FUNCTION_BLOCK fbChamber
VAR_INPUT
END_VAR
VAR_OUTPUT
END_VAR
VAR_IN_OUT
	stControl				: stControl;
	stInOuts 				: stInOuts;
	stParams				: stParamsChamber;
	stChamberTestParams		: stTestParams;
	stTime					: stAircomTimeStruct;	//Struktura czasu
END_VAR
VAR
	//Bloki skalujące
	fbPressureScaller 		:fbAnalogMeasurement;	//Blok skalujący ciśnienie
	fbVoltageScaller	 	:fbAnalogMeasurement;	//Blok skalujący napięcie
	fbCurrentScaller 		:fbAnalogMeasurement;	//Blok skalujący prąd
	iWorkStep : INT;
	//Detekcja prądu
	fbCurrentCheckDelayer	: TON;					//Zwłoka dla wykrywania prądu minimalnego
	//Test EOL
	fbTestTimerEOL			: TON;					//Licznik czasu trwania testu EOL
	bEolTestResult			: BOOL;					//Wynik z testu EOL
	//Test Performance
	fbTestTimerPerformance	: TON;					//Licznik czasu trwania testu Wydajnoiściowego
	bPerfornamceTestResult	: BOOL;					//Wynik z testu Wydajnościowego
	//Test Hour
	fbTestTimerHour	: TON;							//Licznik czasu trwania testu Wydajnoiściowego
	bHourTestResult	: BOOL;							//Wynik z testu Wydajnościowego
	bPressureObtainedHour :BOOL;					//Pierwsza faza zakończona osiągnięto ciśnienie testowe
	//Test Whole
	iWorkStepWhole	: INT;							//Kroki programowe dla testu całościowego
	fbTestTimerWholeI	: TON;							//Licznik czasu I test całkowity
	fbTestTimerWholeII	: TON;							//Licznik czasu II test całkowity
	//Test Under Presure
	bUnderPresureTestResult : BOOL;					//Wynik testu pod ciśnieniem
	rStartUnderPresureLastPresureRecord : REAL;		//Save value of presure before test
	fbUnderPresureTestTimer	: TON;							//Licznik czasu dla tesu pod ciśnieniem
	//Test Cyclic 30
	iCyclicLoopVariable 		: INT;				//Wariable for calculate of cyclic loops
	fbTestTimerCyclic30			: TON;				//Licznik czasu trwania testu cyklicznego 30
	bCyclic30TestResult			: BOOL;				//Wynik testu cyklicznego x30
	fbTestTimerCyclic30On		: TON;				//Timer dla obsługi testu
	bFirstCycle30				: BOOL;				//First cycle indefiner
	//Test Cyclic 70
	fbTestTimerCyclic70			: TON;				//Licznik czasu trwania testu cyklicznego 30
	bCyclic70TestResult			: BOOL;				//Wynik testu cyklicznego x30
	fbTestTimerCyclic70On		: TON;				//Timer dla obsługi testu
	bFirstCycle70				: BOOL;				//First cycle indefiner
	//Zmienne do obsługi zapisu plików
	sData						: STRING;			//Data dopisana do lokalizacji
	sDate						: STRING;			//Data rozpoczęcia testu
	sTime						: STRING;			//Godzina rozpoczęcia testu
	sTestName					: STRING;			//Nazwa Test
	sFirstLine					: STRING;			//Dane do zapisu w pierwszej linijce
	sDataString					: STRING(5000);			//dane z pomiarami
	sDataStringTmp				: STRING(5000);			//dane z pomiarami
	sDataStringTmpSave			: STRING(5000);			//Dane do zapisu
	sActualTestTime				: STRING;			//Aktualny czas testu
	sActualPresure				: STRING;			//Aktualna wartość ciśnienia
	sActualVoltage				: STRING;			//Aktualna wartość napięcia
	sActualCurrent				: STRING;			//Aktualna wartość prądu
	sActualTemperature			: STRING;			//Aktualna wartość temperatury
	fbTestTime					: TON;				//Czas wykonywania testu
	iSaveFileRecords			: INT;				//Aktualnie zapisane rekody do zapisu pliku
	iSaveFileRecordsTmp			: INT;				//Zapisana ilość rekordów w tablicy do zapisu (zmienne skopiowane)
	bCreateFile					: BOOL;				//Wymueszenie utworzenia nowego pliku
	bInsertNewStartRows			: BOOL;				//Wymuszenie wstawienia pierwszych 2 wierszy 
	bSavePerform				: BOOL;				//Wykonaj zapis do pliku
	bCopyArray					: BOOL;				//Przygotowanie buforów do zapisu
	arTmpData					: ARRAY[0..1000] OF STRING;	//Tablica z zmiennymi
	arTmpDataCpy				: ARRAY[0..1000] OF STRING;	//Tablica z zmiennymi skopiowanymi
	fbFileOpen					: FB_FileOpen;		//Funkcja dla otwierania pliku
	fbFileClose					: FB_FileClose;		//Funkcja dla zamknięcia pliku
	fbFileWrite					: FB_FileWrite;		//Funkcja dla zapisu pliku
	sFileNameToSave				: STRING;			//Nazwa do zapisu pliku
	bReadyToWrite				: BOOL;				//Zezwolenie na zapis do pliku
	bReadyToClose				: BOOL;				//Zezwolenie na zamknięcie pliku
	bFileSaveError				: BOOL;				//Błąd podczas tworzenie zapisów
	iSampleRecorder				: INT;				//Obsługa samplingu
	fbTestTimer					: TON;				//Obsługa czasu trwania testu
	sTimeRep					: STRING;			//Zmienna dla obsługi czasu godzina 
	fbRiseEdgeError				: R_TRIG;
	iSaveCalc					: INT;				// zmienna pomocnicza podczas zapisu danych
	bRecordTaker				: BOOL;				//Zmienna dla obsługi zbierania danych
	wRecordCalc					: DWORD;			//Zmienna dla lcizenia czasu testu
	bFileCopy					: BOOL;				//Zmienna wykorzystywana podczas kopiowania plików
	fbFileSave					: fbSaveFiles;		//Save files save
	fbFileSaveCopy				: fbSaveFiles;		//Save files save
	//Zmienne dla obsługi rysowania grafów
	arPlotPresure				: ARRAY[0..1000] OF REAL;
	arPlotVoltage				: ARRAY[0..1000] OF REAL;
	arPlotCurrent				: ARRAY[0..1000] OF REAL;
	iPlotRecordCounter			: INT;
	sStepDescription			: STRING;
	iPlotFilter					: INT;
	sFileCopyCommand			: STRING(1000);
	sTemString					: STRING;
	bTEST: BOOL;
	sDirCopy: STRING;
	sPathCopy:STRING;
	iLastWorkStep: INT;
	fbRestON: TON;
END_VAR

ACT_Background();
CASE iWorkStep OF
 0: 				//Inicalizacja
 	iWorkStep := 5;
	stParams.sErrorDescription :='';
	fbTestTimer(IN:=FALSE);
	stInOuts.bFanON := stInOuts.bPowerON := stInOuts.bEjectPresure40 := stInOuts.bEjectPresure := stInOuts.bBottle40l := stInOuts.bPressureIn := FALSE;
 5:					//Idle
 	sStepDescription := 'Chamber Idle';
	stParams.sTestName:= '';
	stControl.tActualTime := T#40D;
	bUnderPresureTestResult R= bCyclic70TestResult R= bCyclic30TestResult R= bPerfornamceTestResult R= bEolTestResult R= stControl.bStartPerform;
 	IF stControl.bStartPerform AND stControl.iSetTest >= 20 AND stInOuts.rPressure <= stParams.rMinimalPressure THEN
		iWorkStep := 6;
		stControl.tActualTime := stTime.tActualTime;
	ELSIF stControl.bStartPerform AND stControl.iSetTest = nTestType.testEOL AND stInOuts.rPressure <= stParams.rMinimalPressure THEN
		iWorkStep := stControl.iSetTest;
		stControl.bStartPerform := FALSE;
		bInsertNewStartRows := TRUE;
	ELSIF stControl.bStartPerform THEN
		stInOuts.bEjectPresure := TRUE;
		sStepDescription := 'Presure droping';
	END_IF
 6:
 	sStepDescription := 'Wait for bottle 40l';
 	IF stControl.iSetTest = nTestType.testEOL OR NOT stControl.bStartPerform THEN
		iWorkStep := 5;
		stControl.bStartPerform := FALSE;
		stControl.tActualTime := T#40D;
	END_IF
 	IF stControl.bStartAllow THEN
		bInsertNewStartRows := TRUE;
		bUnderPresureTestResult := bCyclic70TestResult := bCyclic30TestResult := bPerfornamceTestResult := bEolTestResult := FALSE;
		iWorkStep := stControl.iSetTest;
		bFirstCycle70 := bFirstCycle30 := TRUE;
		stControl.bStartAllow := FALSE;
		stControl.bStartPerform := FALSE;
	END_IF

 10: 				//EOL Test
 	stParams.sTestName:= 'EOL_Test';
	ACT_EolTest();
	IF bEolTestResult THEN
		iWorkStep := 1000;
	END_IF
 20:				//Performance Test
	stParams.sTestName:= 'Performance_Test';
 	ACT_PerformanceTest();
	IF bPerfornamceTestResult THEN
		iWorkStep := 1000;
	END_IF
 30:				//Hour Test
 	stParams.sTestName:= 'Hour_Test';
 	ACT_HourTest();
	IF bHourTestResult THEN
		iWorkStep := 1000;
	END_IF
 40:				//Whole Test
 	stParams.sTestName:= 'Full_Test';
 	Act_WholeTest();
 50:				//Cyclic x30 Test
 	stParams.sTestName:= 'Cyclic_x30_Test';
 	ACT_Cyclic30Test();
	IF bCyclic30TestResult THEN
		iWorkStep := 1000;
	END_IF
 60:				//Cyclic x70 Test
 	stParams.sTestName:= 'Cyclic_x70_Test';
 	ACT_Cyclic70Test();
	IF bCyclic70TestResult THEN
		iWorkStep := 1000;
	END_IF
 200:				// Błąd
 	stControl.tActualTime := T#40D;
 	fbTestTimer(IN:=FALSE);
	stControl.bStartAllow := stControl.bStartPerform := FALSE;
	IF stInOuts.rPressure >= stParams.rMinimalPressure THEN
		stInOuts.bEjectPresure40 := TRUE;
		sStepDescription := 'Error pressure droping';
	ELSE
		stControl.bTank40Used := FALSE;
		stInOuts.bEjectPresure40 := FALSE;
		sStepDescription := 'Wait for reset';
	END_IF
	
 	bUnderPresureTestResult := bCyclic70TestResult := bCyclic30TestResult := bPerfornamceTestResult := bEolTestResult := stInOuts.bFanON := stInOuts.bPowerON := stInOuts.bEjectPresure := stInOuts.bBottle40l := stInOuts.bPressureIn := FALSE;
 	IF stControl.bResetChamber THEN
		iWorkStep:=0;
		stControl.bResetChamber := FALSE;
		bFileCopy := TRUE;
	END_IF
 1000:				//Przygotowanie komory do następnego testu
 	stInOuts.bEjectPresure40 S= (bPerfornamceTestResult OR bHourTestResult OR bCyclic70TestResult OR bCyclic30TestResult);
	stInOuts.bEjectPresure S= bEolTestResult;
	sStepDescription := 'Presure droping';
 	IF stInOuts.rPressure <= stParams.rMinimalPressure THEN
		stControl.tActualTime := T#40D;
		stInOuts.bEjectPresure40 := stInOuts.bEjectPresure := FALSE;
		iWorkStep := 0;
		bFileCopy := TRUE;
	END_IF
END_CASE

ACTION ACT_Background:
//Obsługa zatrzymania
IF stControl.bChamberBusy AND stControl.bStopPerform THEN
	iWorkStep := 1000;
	stControl.bStopPerform := FALSE;
END_IF
fbRestON(IN:=stControl.bResetChamber,Pt:=T#200MS);
IF fbRestON.Q THEN
	stControl.bResetChamber  := FALSE;
END_IF
//Skalowanie pomiarów Ciśnienia/Napięcia/Prądu
	fbPressureScaller(rIn:=stInOuts.iPressureRaw,stMeasureScalingData:=stParams.stPressureSens,tStalaCzasowa:=T#10MS,rOutFiltered=>stInOuts.rPressure);
	fbVoltageScaller(rIn:=stInOuts.iVoltageRaw,stMeasureScalingData:=stParams.stVoltageSens,tStalaCzasowa:=T#10MS,rOutFiltered=>stInOuts.rVoltage);
	fbCurrentScaller (rIn:=stInOuts.iCurrentRaw,stMeasureScalingData:=stParams.stCurrenteSens,tStalaCzasowa:=T#10MS,rOutFiltered=>stInOuts.rCurrent);
	stInOuts.rTemperature := stInOuts.iTemperature/10;
//Obsługa Safety
IF stInOuts.bSafety	THEN
	stParams.sErrorDescription := 'Emergency button pressed';
	iWorkStep := 200;
END_IF
//Obsługa daty
sData := CONCAT(WORD_TO_STRING(stTime.stTimeStruct.wYear),'_');
sData := CONCAT(sData,WORD_TO_STRING(stTime.stTimeStruct.wMonth));
//Obsługa zbiornika
	stControl.bTank40Used := iWorkStep >= 20; 		//Określenie czy zbiornik 40l jest wykorzystywany
//Obsługa sekwencji
	stControl.bChamberBusy := (iWorkStep >=10);		//Określenie czy komora wykonuje prace
	stControl.bStartPerform R= (iWorkStep > 6);	//Kasowanie wymuszenia staru po rozpoczęciu nowej pracy
//Sprawowanie kontroli nad prądem minimalnym
	fbCurrentCheckDelayer(IN:=stInOuts.bPowerON,PT:=REAL_TO_TIME(stChamberTestParams.rMinimalCurrentCheckDelay*1000));
	IF fbCurrentCheckDelayer.Q AND (stChamberTestParams.rMinimalCurrentLimit > stInOuts.rCurrent) THEN
		stParams.sErrorDescription := 'Minimal current obtain error';
		iWorkStep := 200;
	END_IF
//Zapis Pliku 
sDate := CONCAT(CONCAT(CONCAT(CONCAT(WORD_TO_STRING(stTime.stTimeStruct.wYear),'_'),WORD_TO_STRING(stTime.stTimeStruct.wMonth)),'_'),WORD_TO_STRING(stTime.stTimeStruct.wDay));
sTimeRep := CONCAT(CONCAT(CONCAT(CONCAT(WORD_TO_STRING(stTime.stTimeStruct.wHour),'_'),WORD_TO_STRING(stTime.stTimeStruct.wMinute)),'_'),WORD_TO_STRING(stTime.stTimeStruct.wSecond));	
sDate := CONCAT(CONCAT(sDate,'_'),sTimeRep);
IF stControl.bChamberBusy AND stParams.bSaveToFile THEN
	ACT_DataSampling();
ELSE
	wRecordCalc := 0;
END_IF
IF stControl.bChamberBusy AND (stParams.sErrorDescription = '') THEN
	ACT_GraphWriter();
	sStepDescription := 'Work in progress';
ELSIF iPlotRecordCounter <> 0 THEN
	iPlotRecordCounter := 0;
	MEMSET(destAddr:=ADR(arPlotPresure),fillByte:=16#00,n:=SIZEOF(arPlotPresure[0])*1000);
	MEMSET(destAddr:=ADR(arPlotVoltage),fillByte:=16#00,n:=SIZEOF(arPlotVoltage[0])*1000);
	MEMSET(destAddr:=ADR(arPlotCurrent),fillByte:=16#00,n:=SIZEOF(arPlotCurrent[0])*1000);
ELSIF NOT stControl.bChamberBusy AND stParams.sErrorDescription = '' THEN
	sStepDescription := 'Idle';
ELSIF stParams.sErrorDescription <> '' THEN
	sStepDescription := 'Chamber Error';
END_IF
//Timer dla obsługi aktualnego czasu
fbTestTime(IN:=stControl.bChamberBusy,PT:=T#5D);
//Wyniki z testów
stControl.bChamberResoult := bUnderPresureTestResult OR bCyclic70TestResult OR bCyclic30TestResult OR bPerfornamceTestResult OR bEolTestResult;
END_ACTION

ACTION ACT_Cyclic30Test:
fbTestTimer(IN:=stINOuts.bPowerON,PT:=T#10D);
IF fbTestTimerCyclic30On.Q OR bFirstCycle30 THEN
	stInOuts.bEjectPresure40 := stInOuts.bEjectPresure := stInOuts.bPressureIn := FALSE;
	stInOuts.bBottle40l := stInOuts.bFanON := stInOuts.bPowerON := TRUE;
	fbTestTimerCyclic30(IN:= stInOuts.bPowerON,PT:=REAL_TO_TIME(stChamberTestParams.rTestCycle30LimitTime*1000));
	IF (fbTestTimerPerformance.Q AND stChamberTestParams.rPresureToObtainCycle30Test >= stInOuts.rPressure) THEN
		iWorkStep:= 200;
		stInOuts.bFanON := stInOuts.bPowerON := FALSE;
		stInOuts.bEjectPresure40 := stInOuts.bEjectPresure := TRUE;
		stParams.sErrorDescription := 'Compressor did not obtain set pressure in limited time';
		bPerfornamceTestResult := FALSE;
		fbTestTimerPerformance(IN:=FALSE);
	ELSIF (stChamberTestParams.rCurrentLimitCycle30 < stInOuts.rCurrent) THEN
		iWorkStep:= 200;
		stInOuts.bFanON := stInOuts.bPowerON := FALSE;
		stInOuts.bEjectPresure40 := stInOuts.bEjectPresure := TRUE;
		stParams.sErrorDescription := 'Current to high';
		bPerfornamceTestResult := FALSE;
		fbTestTimerPerformance(IN:=FALSE);
	END_IF
	IF fbTestTimerPerformance.Q AND stChamberTestParams.rPresureToObtainCycle30Test <= stInOuts.rPressure THEN
		iCyclicLoopVariable := iCyclicLoopVariable + 1;
		bFirstCycle30 := FALSE;
		stInOuts.bEjectPresure40 := stInOuts.bEjectPresure := TRUE;
		stInOuts.bPowerON := FALSE;
		fbTestTimerCyclic30On(IN:=FALSE);
		fbTestTimerCyclic30(IN:=FALSE);
		stInOuts.bPowerON := FALSE;
		IF iCyclicLoopVariable >=30 THEN
			bCyclic30TestResult := TRUE;
			iCyclicLoopVariable := 0;
			bFirstCycle30:= TRUE;
		END_IF
	END_IF
ELSE
	fbTestTimerCyclic30On(IN:=TRUE,PT:=REAL_TO_TIME(stChamberTestParams.rTestCycle30CoolingTime*1000));
END_IF
END_ACTION

ACTION ACT_Cyclic70Test:
fbTestTimer(IN:=stINOuts.bPowerON,PT:=T#10D);
IF fbTestTimerCyclic70On.Q OR bFirstCycle70 THEN
	stInOuts.bEjectPresure40 := stInOuts.bEjectPresure := stInOuts.bPressureIn := FALSE;
	stInOuts.bBottle40l := stInOuts.bFanON := stInOuts.bPowerON := TRUE;
	fbTestTimerCyclic70(IN:= stInOuts.bPowerON,PT:=REAL_TO_TIME(stChamberTestParams.rTestCycle70LimitTime*1000));
	IF (fbTestTimerPerformance.Q AND stChamberTestParams.rPresureToObtainCycle70Test >= stInOuts.rPressure) THEN
		iWorkStep:= 200;
		stInOuts.bFanON := stInOuts.bPowerON := FALSE;
		stInOuts.bEjectPresure40 := stInOuts.bEjectPresure := TRUE;
		stParams.sErrorDescription := 'Compressor did not obtain set pressure in limited time';
		bPerfornamceTestResult := FALSE;
		fbTestTimerPerformance(IN:=FALSE);
	ELSIF (stChamberTestParams.rCurrentLimitCycle70 < stInOuts.rCurrent) THEN
		iWorkStep:= 200;
		stInOuts.bFanON := stInOuts.bPowerON := FALSE;
		stInOuts.bEjectPresure40 := stInOuts.bEjectPresure := TRUE;
		stParams.sErrorDescription := 'Current to high';
		bPerfornamceTestResult := FALSE;
		fbTestTimerPerformance(IN:=FALSE);
	END_IF
	IF fbTestTimerPerformance.Q AND stChamberTestParams.rPresureToObtainCycle70Test <= stInOuts.rPressure THEN
		iCyclicLoopVariable := iCyclicLoopVariable + 1;
		bFirstCycle70 := FALSE;
		stInOuts.bEjectPresure40 := stInOuts.bEjectPresure := TRUE;
		stInOuts.bPowerON := FALSE;
		fbTestTimerCyclic70On(IN:=FALSE);
		fbTestTimerCyclic70(IN:=FALSE);
		stInOuts.bPowerON := FALSE;
		IF iCyclicLoopVariable >=30 THEN
			bCyclic70TestResult := TRUE;
			iCyclicLoopVariable := 0;
			bFirstCycle70:= TRUE;
		END_IF
	END_IF
ELSE
	fbTestTimerCyclic70On(IN:=TRUE,PT:=REAL_TO_TIME(stChamberTestParams.rTestCycle30CoolingTime*1000));
END_IF
END_ACTION

ACTION ACT_DataSampling:
IF iWorkStep <> iLastWorkStep THEN
	iLastWorkStep := iWorkStep;
	wRecordCalc := 0;
END_IF
wRecordCalc := wRecordCalc +1;
//Przygotowywanie zmiennych nagłówkowych
IF bInsertNewStartRows AND stParams.sTestName <> '' THEN
	//Przygotowanie ścieżki pliku z nazwą
	sFileNameToSave:= '';
	sFileNameToSave:= CONCAT(sFileNameToSave,sDate);
	sFileNameToSave:= CONCAT(sFileNameToSave,'_');
	sFileNameToSave:= CONCAT(sFileNameToSave,stParams.sChamberName);
	sFileNameToSave:= CONCAT(sFileNameToSave,'_');
	sFileNameToSave:= CONCAT(sFileNameToSave,sTestName);
	sFileNameToSave:= CONCAT(sFileNameToSave,'_');
	sFileNameToSave:= CONCAT(sFileNameToSave,stParams.sTestName);
	sFileNameToSave:= CONCAT(sFileNameToSave,'.csv');
	bInsertNewStartRows := FALSE;
	//Tworzenie nagłówków 
	sDataStringTmp := CONCAT(sDate,',');
	sDataStringTmp := CONCAT(sDataStringTmp,stParams.sChamberName);
	sDataStringTmp := CONCAT(sDataStringTmp,',');
	sDataStringTmp := CONCAT(sDataStringTmp,stParams.sFileName);
	sDataStringTmp := CONCAT(sDataStringTmp,',');
	sDataStringTmp := CONCAT(sDataStringTmp,sTestName);
	sDataStringTmp := CONCAT(sDataStringTmp,'$R');
	sDataStringTmp := CONCAT(sDataStringTmp,'Czas [s],Prąd [A],Ciśnienie [bar],Napięcie [V],Temperatura [°C]$R');
	sDataString := sDataStringTmp;
	iSaveFileRecords := 2;
END_IF
//Cykliczne przygotowyawanie zmiennych
IF stParams.sErrorDescription = '' THEN
	iSampleRecorder := iSampleRecorder + 1;
	bRecordTaker := (*iSampleRecorder >= 1;*)(iSampleRecorder >= stParams.iSampleTime0_150/10 AND  wRecordCalc  <=  15) OR (iSampleRecorder >= stParams.iSampleTime0_1/10 AND  wRecordCalc  > 15 AND  wRecordCalc  <=  100) 
		OR (iSampleRecorder >= stParams.iSampleTime1_x/10 AND  wRecordCalc  >  100);
	IF bRecordTaker THEN
		sActualTestTime 	:= REAL_TO_STRING(TIME_TO_REAL(fbTestTime.ET)/1000);
		sActualPresure 		:= REAL_TO_STRING(stInOuts.rPressure);					//Przepisanie wartości ciśnienia
		sActualVoltage 		:= REAL_TO_STRING(stInOuts.rVoltage);					//Przepisanie wartości napięcia
		sActualCurrent 		:= REAL_TO_STRING(stInOuts.rCurrent);					//Przepisanie wartości prądu
		sActualTemperature 	:= REAL_TO_STRING(stInOuts.rTemperature);											//Przepisanie wartości temperatury
		//Przygotowanie zmiennych cyklicznych do zapisu oraz przemieszczenie danych do bufora
		sDataStringTmp 		:= CONCAT(sActualTestTime,',');					//Zapisanie aktualnego czasu 
		sDataStringTmp 		:= CONCAT(sDataStringTmp,sActualCurrent);			//Dopisanie wartości prądu
		sDataStringTmp 		:= CONCAT(sDataStringTmp,',');						//Przypisanie odstępu format CSV
		sDataStringTmp 		:= CONCAT(sDataStringTmp,sActualPresure);			//Dopisanie wartości ciśnienia
		sDataStringTmp 		:= CONCAT(sDataStringTmp,',');						//Przypisanie odstępu format CSV
		sDataStringTmp 		:= CONCAT(sDataStringTmp,sActualVoltage);			//Dopisanie wartości napięcia
		sDataStringTmp 		:= CONCAT(sDataStringTmp,',');						//Przypisanie odstępu format CSV
		sDataStringTmp 		:= CONCAT(sDataStringTmp,sActualTemperature);		//Dopisanie wartości temperatury
		sDataStringTmp 		:= CONCAT(sDataStringTmp,'$R');						//Dopisanie znaku enter
		CONCAT2(pSrcString1:=ADR(sDataString),pSrcString2:=ADR(sDataStringTmp),pDstString:=ADR(sDataString),nDstSize:=SIZEOF(sDataString));
		iSaveFileRecords 	:= iSaveFileRecords + 1;
		iSampleRecorder 	:= 0;
	END_IF
END_IF
//Wykonanie zapisu oraz uporzątkowanie zmiennych/buforów
fbRiseEdgeError(CLK:=(stParams.sErrorDescription <> '' OR iWorkStep = 1000));
fbFileSave.bExecute S= ((iSaveFileRecords >= stParams.iSaveEveryRecords) OR fbRiseEdgeError.Q ) AND NOT fbFileSave.bBusy;
fbFileSaveCopy.bExecute S= ((iSaveFileRecords >= stParams.iSaveEveryRecords) OR fbRiseEdgeError.Q ) AND NOT fbFileSave.bBusy;
IF fbFileSave.bDone AND fbFileSave.bDone THEN
	iSaveFileRecords := 0;
	fbFileSave.bExecute R= TRUE;
	fbFileSaveCopy.bExecute R= TRUE;
	sDataString := '';
END_IF
fbFileSave(
	sFileNameToSave:=sFileNameToSave,
	sDataStringTmpSave:=sDataString,
	sFileDirectory:=CONCAT(stParams.sFileDirectory,sData));
fbFileSaveCopy(
	sFileNameToSave:=sFileNameToSave,
	sDataStringTmpSave:=sDataString,
	sFileDirectory:=CONCAT(stParams.sFileCopyLocation,sData));
END_ACTION

ACTION ACT_EolTest:
fbTestTimer(IN:=stINOuts.bPowerON,PT:=T#10D);
stInOuts.bEjectPresure40 := stInOuts.bEjectPresure := stInOuts.bBottle40l := stInOuts.bPressureIn := FALSE;
stInOuts.bFanON := stInOuts.bPowerON := TRUE;
fbTestTimerEOL(IN:= stInOuts.bPowerON,PT:=REAL_TO_TIME(stChamberTestParams.rTestEolLimitTime*1000));
IF fbTestTimerEOL.Q THEN
	iWorkStep:= 200;
	stInOuts.bFanON := stInOuts.bPowerON := FALSE;
	stInOuts.bEjectPresure := TRUE;
	stParams.sErrorDescription := 'Compressor did not obtain set pressure in limited time';
	bEolTestResult := FALSE;
	fbTestTimerEOL(IN:=FALSE);
END_IF
IF stChamberTestParams.rPresureToObtainEOLTest < stInOuts.rPressure THEN
	bEolTestResult := TRUE;
	fbTestTimerEOL(IN:=FALSE);
END_IF
END_ACTION

ACTION ACT_GraphWriter:
iPlotFilter := iPlotFilter + 1;
IF iPlotFilter >= 5 THEN
	arPlotPresure[iPlotRecordCounter] := stInOuts.rPressure;
	arPlotVoltage[iPlotRecordCounter] := stInOuts.rVoltage;
	arPlotCurrent[iPlotRecordCounter] := stInOuts.rCurrent;
	iPlotRecordCounter := iPlotRecordCounter + 1;
	iPlotFilter := 0;
	IF iPlotRecordCounter >= 500 THEN
		iPlotRecordCounter := 0;
		MEMSET(destAddr:=ADR(arPlotPresure),fillByte:=16#00,n:=SIZEOF(arPlotPresure[0])*1000);
		MEMSET(destAddr:=ADR(arPlotVoltage),fillByte:=16#00,n:=SIZEOF(arPlotVoltage[0])*1000);
		MEMSET(destAddr:=ADR(arPlotCurrent),fillByte:=16#00,n:=SIZEOF(arPlotCurrent[0])*1000);
	END_IF
END_IF
END_ACTION

ACTION ACT_HourTest:
fbTestTimer(IN:=stINOuts.bPowerON,PT:=T#10D);
stInOuts.bEjectPresure40 := stInOuts.bEjectPresure := stInOuts.bPressureIn := FALSE;
stInOuts.bBottle40l := stInOuts.bFanON := stInOuts.bPowerON := TRUE;
fbTestTimerHour(IN:= (stChamberTestParams.rPressureToObtainHourTest<=stInOuts.rPressure),PT:=REAL_TO_TIME(stChamberTestParams.rTestHourTime*1000));
bPressureObtainedHour S= (stChamberTestParams.rPressureToObtainHourTest<=stInOuts.rPressure);
IF bPressureObtainedHour AND ABS(stInOuts.rPressure-stChamberTestParams.rPressureToObtainHourTest) > stChamberTestParams.rTestHourPressureMaximalTolerance THEN
	iWorkStep:= 200;
	stInOuts.bFanON := stInOuts.bPowerON := FALSE;
	stInOuts.bEjectPresure40 := stInOuts.bEjectPresure := TRUE;
	stParams.sErrorDescription := 'Pressure deviation too high';
	bHourTestResult := FALSE;
	fbTestTimerHour(IN:= FALSE);
END_IF
IF fbTestTimerPerformance.Q THEN
	bHourTestResult := TRUE;
	bPressureObtainedHour R= TRUE;
	fbTestTimerHour(IN:= FALSE);
END_IF
END_ACTION

ACTION ACT_PerformanceTest:
fbTestTimer(IN:=stINOuts.bPowerON,PT:=T#10D);
stInOuts.bEjectPresure40 := stInOuts.bEjectPresure := stInOuts.bPressureIn := FALSE;
stInOuts.bBottle40l := stInOuts.bFanON := stInOuts.bPowerON := TRUE;
fbTestTimerPerformance(IN:= stInOuts.bPowerON,PT:=REAL_TO_TIME(stChamberTestParams.rTest300SecTime*1000));
IF (fbTestTimerPerformance.Q AND stChamberTestParams.rPresureToObtainPerformanceTest >= stInOuts.rPressure) THEN
	iWorkStep:= 200;
	stInOuts.bFanON := stInOuts.bPowerON := FALSE;
	stInOuts.bEjectPresure40 := stInOuts.bEjectPresure := TRUE;
	stParams.sErrorDescription := 'Compressor did not obtain set pressure in limited time';
	bPerfornamceTestResult := FALSE;
	fbTestTimerPerformance(IN:=FALSE);
ELSIF (stChamberTestParams.rCurrentLimitPerformacneTest < stInOuts.rCurrent) THEN
	iWorkStep:= 200;
	stInOuts.bFanON := stInOuts.bPowerON := FALSE;
	stInOuts.bEjectPresure40 := stInOuts.bEjectPresure := TRUE;
	stParams.sErrorDescription := 'Current to high';
	bPerfornamceTestResult := FALSE;
	fbTestTimerPerformance(IN:=FALSE);
END_IF
IF fbTestTimerPerformance.Q AND stChamberTestParams.rPresureToObtainPerformanceTest <= stInOuts.rPressure THEN
	bPerfornamceTestResult := TRUE;
	fbTestTimerPerformance(IN:=FALSE);
END_IF
END_ACTION

ACTION ACT_TestUnderPressure:
fbTestTimer(IN:=stINOuts.bPowerON,PT:=T#10D);
IF stInOuts.rPressure < (stChamberTestParams.rTestUnderPresureSetPresure - stChamberTestParams.rTestUnderPresureCloseTolerance) THEN
	stInOuts.bEjectPresure40 := stInOuts.bEjectPresure := FALSE;
	stInOuts.bPressureIn := stInOuts.bBottle40l := TRUE;
ELSE
	stInOuts.bPressureIn := FALSE;
END_IF
IF ABS(stInOuts.rPressure - stChamberTestParams.rTestUnderPresureSetPresure) < stChamberTestParams.rTestUnderPresureStartTolerance AND NOT stInOuts.bPressureIn THEN
	stInOuts.bPowerON := TRUE;
	rStartUnderPresureLastPresureRecord := stInOuts.rPressure;
END_IF

IF stInOuts.bPowerON THEN
	fbUnderPresureTestTimer(IN:=TRUE,PT:=REAL_TO_TIME(stChamberTestParams.rTestUnderPresureTime*1000));
	IF (stInOuts.rPressure - stChamberTestParams.rTestUnderPresureSetPresure) > stChamberTestParams.rTestUnderPresureMinimalIncrease THEN
		bUnderPresureTestResult := TRUE;
	ELSIF fbUnderPresureTestTimer.Q THEN
		iWorkStep:= 200;
		stInOuts.bFanON := stInOuts.bPowerON := FALSE;
		stInOuts.bEjectPresure40 := stInOuts.bEjectPresure := TRUE;
		stParams.sErrorDescription := 'Start under presure failt to obtain presure increase in definied time';
		bUnderPresureTestResult := FALSE;
		fbTestTimerPerformance(IN:=FALSE);
	END_IF
END_IF
END_ACTION

ACTION ACT_WholeTest:
CASE iWorkStepWhole OF 
	0:	//Test wydajnościowy
		ACT_PerformanceTest();
		IF bPerfornamceTestResult THEN
			iWorkStepWhole := 5;
		END_IF
	5:
		stInOuts.bEjectPresure40 S= (bPerfornamceTestResult OR bHourTestResult);
		stInOuts.bEjectPresure S= bEolTestResult;
		IF stInOuts.rPressure <= stParams.rMinimalPressure THEN
			stInOuts.bEjectPresure40 := stInOuts.bEjectPresure := FALSE;
			iWorkStepWhole := 10;
		END_IF
	10:	//Oczekiwanie 
		fbTestTimerWholeI(IN:=TRUE,PT:=REAL_TO_TIME(stChamberTestParams.rTestCoolingTimeFullStepI*1000));
		IF fbTestTimerWholeI.Q THEN
			iWorkStepWhole := 20;
			fbTestTimerWholeI(IN:=FALSE);
		END_IF
	20:	//Test godzinny
		ACT_HourTest();
		IF bHourTestResult THEN
			iWorkStepWhole := 25;
		END_IF
	25: //Test pod ciśnieniem
		ACT_TestUnderPressure();
		IF bUnderPresureTestResult THEN
			iWorkStepWhole := 30;
		END_IF
	30:
		stInOuts.bEjectPresure40 S= (bPerfornamceTestResult OR bHourTestResult);
		stInOuts.bEjectPresure S= bEolTestResult;
		IF stInOuts.rPressure <= stParams.rMinimalPressure THEN
			stInOuts.bEjectPresure40 := stInOuts.bEjectPresure := FALSE;
			iWorkStepWhole := 35;
		END_IF
	35:	//Oczekiwanie II
		fbTestTimerWholeII(IN:=TRUE,PT:=REAL_TO_TIME(stChamberTestParams.rTestCoolingTimeFullStepII*1000));
		IF fbTestTimerWholeII.Q THEN
			iWorkStepWhole := 40;
			fbTestTimerWholeII(IN:=FALSE);
		END_IF
	40:
		ACT_PerformanceTest();
		IF bPerfornamceTestResult THEN
			iWorkStep:=1000;
			iWorkStepWhole := 0;
		END_IF
	



END_CASE
END_ACTION

END_FUNCTION_BLOCK

(* stored: Version 1.1.0.1, ProductVersion 3.1.4024.12
   POU fbChamber: Id {92018890-bba3-4a0b-9c46-efc95a910be5}, SpecialFunc None
   Folder Tests: Id {f2c98301-b4b3-4559-b309-e9009caa9302}
   Action ACT_Background: Id {26932ffc-0ce0-4424-833b-d11150f7d951}
   Action ACT_Cyclic30Test: Id {6c4769a7-ccce-4c82-a5e6-dc70a100a96b}
   Action ACT_Cyclic70Test: Id {bf6d1270-e215-4f8f-82b2-fb34b284a109}
   Action ACT_DataSampling: Id {ea2532f0-ebff-4831-ad56-5d5bba884596}
   Action ACT_EolTest: Id {3e8dafe0-fbc8-4fbd-a9f0-c41b276ef449}
   Action ACT_GraphWriter: Id {ca0bbc37-a33f-4a95-ad90-74dcb0d0d1c6}
   Action ACT_HourTest: Id {02181811-977a-4078-b3e9-3f316e52df8f}
   Action ACT_PerformanceTest: Id {fd61ae1f-5b08-4c39-a2da-c86c8c4f2eb3}
   Action ACT_TestUnderPressure: Id {2038a382-89b2-4823-97f1-7eeed3d570ce}
   Action ACT_WholeTest: Id {27d190bc-b86a-4499-ba6e-4a762a3fc3bc} *)
